{attribute 'GeneratedUsingTerminal: EL2564-0000-0016'}
{attribute addProperty BoxType "EL2564-0000-0016"}
{attribute addProperty Id "PWM_Inputs_Channel_1AT %I*PWM_Inputs_Channel_304DC2453PWM_Inputs_Channel_2AT %I*PWM_Inputs_Channel_304DC2453PWM_Inputs_Channel_3AT %I*PWM_Inputs_Channel_304DC2453PWM_Inputs_Channel_4AT %I*PWM_Inputs_Channel_304DC2453PWM_Outputs_Channel_1AT %Q*PWM_Outputs_Channel_D6F04FBD2PWM_Outputs_Channel_2AT %Q*PWM_Outputs_Channel_D6F04FBD2PWM_Outputs_Channel_3AT %Q*PWM_Outputs_Channel_D6F04FBD2PWM_Outputs_Channel_4AT %Q*PWM_Outputs_Channel_D6F04FBD2WcStateAT %I*WcState_9091E0EB2InfoDataAT %I*InfoData_94A18F5E2"}
{attribute addProperty CRC "1238969800"}
{attribute addProperty Size "24"}
TYPE EL2564_49D92DC8 EXTENDS EtcSlaveTerminalBase_947E5A46 :
STRUCT
	{attribute addProperty Name "PWM_Inputs_Channel_1"}
	PWM_Inputs_Channel_1 : PWM_Inputs_Channel_304DC245;
	{attribute addProperty Name "PWM_Inputs_Channel_2"}
	PWM_Inputs_Channel_2 : PWM_Inputs_Channel_304DC245;
	{attribute addProperty Name "PWM_Inputs_Channel_3"}
	PWM_Inputs_Channel_3 : PWM_Inputs_Channel_304DC245;
	{attribute addProperty Name "PWM_Inputs_Channel_4"}
	PWM_Inputs_Channel_4 : PWM_Inputs_Channel_304DC245;
	{attribute addProperty Name "PWM_Outputs_Channel_1"}
	PWM_Outputs_Channel_1 : PWM_Outputs_Channel_D6F04FBD;
	{attribute addProperty Name "PWM_Outputs_Channel_2"}
	PWM_Outputs_Channel_2 : PWM_Outputs_Channel_D6F04FBD;
	{attribute addProperty Name "PWM_Outputs_Channel_3"}
	PWM_Outputs_Channel_3 : PWM_Outputs_Channel_D6F04FBD;
	{attribute addProperty Name "PWM_Outputs_Channel_4"}
	PWM_Outputs_Channel_4 : PWM_Outputs_Channel_D6F04FBD;
	{attribute addProperty Name "WcState"}
	WcState : WcState_9091E0EB;
	{attribute addProperty Name "InfoData"}
	InfoData : InfoData_94A18F5E;
END_STRUCT
END_TYPE

(* stored: Version 1.2.0.0, ProductVersion 3.1.4024.9
   DUT EL2564_49D92DC8: Id {96663606-0d3f-4204-84e9-5434fac33598} *)
